ABB RAPID module: test02_001.prg

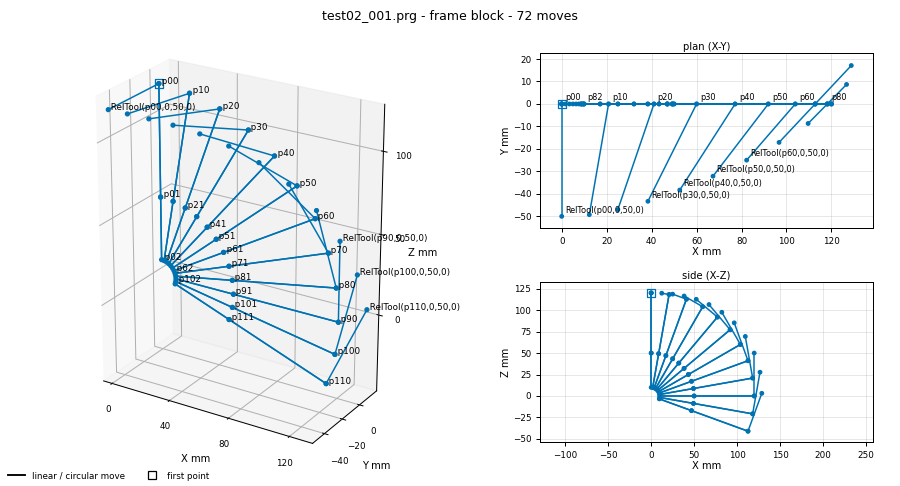
[picture p0: tool path of test02_001.prg in frame block, 72 of 87 moves have a stored position in this frame; points joined in program order, loops and branches not executed]
MODULE MainModule

	! test02_001

	! variables
	TASK PERS tooldata drill := [FALSE, [[300,-260,280], [0,0,0,1]], [1,[0,0,0.001],[1,0,0,0],0,0,0]];
	TASK PERS wobjdata block := [TRUE, TRUE, "", [[0,0,150], [1,0,0,0]], [[0,0,0], [1,0,0,0]]];
	TASK PERS speeddata rate := [3, 500, 5000, 1000];

	! targets
	VAR jointtarget j0 := [[-90,0,0,90,90,0], [9E9,9E9,9E9,9E9,9E9,9E9]];
	VAR jointtarget j1 := [[-41,0,0,0,90,0], [9E9,9E9,9E9,9E9,9E9,9E9]];
	VAR robtarget p00 := [[2.20429143688028E-14,0,120], [0,1,0,-9.18454765366783E-17], [0,0,0,0], [9E9,9E9,9E9,9E9,9E9,9E9]];
	VAR robtarget p01 := [[9.18454765366783E-15,0,50], [0,1,0,-9.18454765366783E-17], [0,0,0,0], [9E9,9E9,9E9,9E9,9E9,9E9]];
	VAR robtarget p02 := [[1.83690953073357E-15,0,10], [0,1,0,-9.18454765366783E-17], [0,0,0,0], [9E9,9E9,9E9,9E9,9E9,9E9]];
	VAR robtarget p10 := [[20.8377813200316,-1.2490009027033E-15,118.176930361465], [0.00759612349389579,0.992403876506124,-0.0868240888334661,-0.086824088833467], [0,0,0,0], [9E9,9E9,9E9,9E9,9E9,9E9]];
	VAR robtarget p11 := [[8.68240888334652,-5.20417042793042E-16,49.2403876506104], [0.00759612349389579,0.992403876506124,-0.0868240888334661,-0.086824088833467], [0,0,0,0], [9E9,9E9,9E9,9E9,9E9,9E9]];
	VAR robtarget p12 := [[1.7364817766693,-1.04083408558608E-16,9.84807753012208], [0.00759612349389579,0.992403876506124,-0.0868240888334661,-0.086824088833467], [0,0,0,0], [9E9,9E9,9E9,9E9,9E9,9E9]];
	VAR robtarget p20 := [[41.0424171990802,-1.66533453693773E-15,112.763114494309], [0.0301536896070456,0.969846310392959,-0.171010071662836,-0.171010071662835], [0,0,0,0], [9E9,9E9,9E9,9E9,9E9,9E9]];
	VAR robtarget p21 := [[17.1010071662834,-6.93889390390723E-16,46.9846310392954], [0.0301536896070456,0.969846310392959,-0.171010071662836,-0.171010071662835], [0,0,0,0], [9E9,9E9,9E9,9E9,9E9,9E9]];
	VAR robtarget p22 := [[3.42020143325669,-1.38777878078145E-16,9.39692620785909], [0.0301536896070456,0.969846310392959,-0.171010071662836,-0.171010071662835], [0,0,0,0], [9E9,9E9,9E9,9E9,9E9,9E9]];
	VAR robtarget p30 := [[60.0000000000001,-6.66133814775094E-15,103.923048454133], [0.0669872981077809,0.933012701892218,-0.249999999999999,-0.25], [0,0,0,0], [9E9,9E9,9E9,9E9,9E9,9E9]];
	VAR robtarget p31 := [[25,-2.77555756156289E-15,43.3012701892219], [0.0669872981077809,0.933012701892218,-0.249999999999999,-0.25], [0,0,0,0], [9E9,9E9,9E9,9E9,9E9,9E9]];
	VAR robtarget p32 := [[5,-5.55111512312578E-16,8.66025403784439], [0.0669872981077809,0.933012701892218,-0.249999999999999,-0.25], [0,0,0,0], [9E9,9E9,9E9,9E9,9E9,9E9]];
	VAR robtarget p40 := [[77.1345131623847,6.66133814775094E-15,91.9253331742773], [0.116977778440511,0.883022221559491,-0.32139380484327,-0.32139380484327], [0,0,0,0], [9E9,9E9,9E9,9E9,9E9,9E9]];
	VAR robtarget p41 := [[32.139380484327,2.77555756156289E-15,38.3022221559489], [0.116977778440511,0.883022221559491,-0.32139380484327,-0.32139380484327], [0,0,0,0], [9E9,9E9,9E9,9E9,9E9,9E9]];
	VAR robtarget p42 := [[6.4278760968654,5.55111512312578E-16,7.66044443118978], [0.116977778440511,0.883022221559491,-0.32139380484327,-0.32139380484327], [0,0,0,0], [9E9,9E9,9E9,9E9,9E9,9E9]];
	VAR robtarget p50 := [[91.9253331742774,9.99200722162641E-15,77.1345131623847], [0.17860619515673,0.82139380484327,-0.383022221559489,-0.383022221559489], [0,0,0,0], [9E9,9E9,9E9,9E9,9E9,9E9]];
	VAR robtarget p51 := [[38.3022221559489,4.16333634234434E-15,32.139380484327], [0.17860619515673,0.82139380484327,-0.383022221559489,-0.383022221559489], [0,0,0,0], [9E9,9E9,9E9,9E9,9E9,9E9]];
	VAR robtarget p52 := [[7.66044443118978,8.32667268468867E-16,6.4278760968654], [0.17860619515673,0.82139380484327,-0.383022221559489,-0.383022221559489], [0,0,0,0], [9E9,9E9,9E9,9E9,9E9,9E9]];
	VAR robtarget p60 := [[103.923048454133,1.33226762955019E-14,60], [0.25,0.75,-0.433012701892219,-0.433012701892219], [0,0,0,0], [9E9,9E9,9E9,9E9,9E9,9E9]];
	VAR robtarget p61 := [[43.3012701892219,5.55111512312578E-15,25], [0.25,0.75,-0.433012701892219,-0.433012701892219], [0,0,0,0], [9E9,9E9,9E9,9E9,9E9,9E9]];
	VAR robtarget p62 := [[8.66025403784439,1.11022302462516E-15,5], [0.25,0.75,-0.433012701892219,-0.433012701892219], [0,0,0,0], [9E9,9E9,9E9,9E9,9E9,9E9]];
	VAR robtarget p70 := [[112.763114494309,6.66133814775094E-15,41.0424171990802], [0.328989928337166,0.671010071662834,-0.469846310392954,-0.469846310392954], [0,0,0,0], [9E9,9E9,9E9,9E9,9E9,9E9]];
	VAR robtarget p71 := [[46.9846310392954,2.77555756156289E-15,17.1010071662834], [0.328989928337166,0.671010071662834,-0.469846310392954,-0.469846310392954], [0,0,0,0], [9E9,9E9,9E9,9E9,9E9,9E9]];
	VAR robtarget p72 := [[9.39692620785909,5.55111512312578E-16,3.42020143325669], [0.328989928337166,0.671010071662834,-0.469846310392954,-0.469846310392954], [0,0,0,0], [9E9,9E9,9E9,9E9,9E9,9E9]];
	VAR robtarget p80 := [[118.176930361465,3.7470027081099E-15,20.8377813200317], [0.413175911166535,0.586824088833465,-0.492403876506104,-0.492403876506104], [0,0,0,0], [9E9,9E9,9E9,9E9,9E9,9E9]];
	VAR robtarget p81 := [[49.2403876506104,1.56125112837913E-15,8.68240888334652], [0.413175911166535,0.586824088833465,-0.492403876506104,-0.492403876506104], [0,0,0,0], [9E9,9E9,9E9,9E9,9E9,9E9]];
	VAR robtarget p82 := [[9.84807753012208,3.12250225675825E-16,1.7364817766693], [0.413175911166535,0.586824088833465,-0.492403876506104,-0.492403876506104], [0,0,0,0], [9E9,9E9,9E9,9E9,9E9,9E9]];
	VAR robtarget p90 := [[120,-8.99826150854451E-31,-1.46952762458685E-14], [0.5,0.5,-0.5,-0.5], [0,0,0,0], [9E9,9E9,9E9,9E9,9E9,9E9]];
	VAR robtarget p91 := [[50,-3.74927562856021E-31,-6.12303176911188E-15], [0.5,0.5,-0.5,-0.5], [0,0,0,0], [9E9,9E9,9E9,9E9,9E9,9E9]];
	VAR robtarget p92 := [[10,-7.49855125712043E-32,-1.22460635382238E-15], [0.5,0.5,-0.5,-0.5], [0,0,0,0], [9E9,9E9,9E9,9E9,9E9,9E9]];
	VAR robtarget p100 := [[118.176930361465,-1.66533453693773E-15,-20.8377813200316], [0.586824088833465,0.413175911166535,-0.492403876506104,-0.492403876506104], [0,0,0,0], [9E9,9E9,9E9,9E9,9E9,9E9]];
	VAR robtarget p101 := [[49.2403876506104,-6.93889390390723E-16,-8.68240888334652], [0.586824088833465,0.413175911166535,-0.492403876506104,-0.492403876506104], [0,0,0,0], [9E9,9E9,9E9,9E9,9E9,9E9]];
	VAR robtarget p102 := [[9.84807753012208,-1.38777878078145E-16,-1.7364817766693], [0.586824088833465,0.413175911166535,-0.492403876506104,-0.492403876506104], [0,0,0,0], [9E9,9E9,9E9,9E9,9E9,9E9]];
	VAR robtarget p110 := [[112.763114494309,-3.33066907387547E-15,-41.0424171990803], [0.671010071662834,0.328989928337166,-0.469846310392954,-0.469846310392954], [0,0,0,0], [9E9,9E9,9E9,9E9,9E9,9E9]];
	VAR robtarget p111 := [[46.9846310392954,-1.38777878078145E-15,-17.1010071662834], [0.671010071662834,0.328989928337166,-0.469846310392954,-0.469846310392954], [0,0,0,0], [9E9,9E9,9E9,9E9,9E9,9E9]];
	VAR robtarget p112 := [[9.39692620785908,-2.77555756156289E-16,-3.42020143325669], [0.671010071662834,0.328989928337166,-0.469846310392954,-0.469846310392954], [0,0,0,0], [9E9,9E9,9E9,9E9,9E9,9E9]];

	! drilling instructions
	PROC main()
		ConfL\Off;
		SingArea\Wrist;

		TPWrite("This is: test02_001");
		TPWrite("Check block and drill");
		MoveAbsJ j0, v100, z5, tool0;
		MoveAbsJ j1, v100, z5, tool0;

		TPWrite("Drilling hole 1 of 12!");
		MoveL p00, v100, z30, drill\WObj:=block;
		MoveL p01, v100, z5, drill\WObj:=block;
		MoveL p02, rate, fine, drill\WObj:=block;
		MoveL p01, rate, fine, drill\WObj:=block;
		MoveL p00, v100, z30, drill\WObj:=block;
		MoveL RelTool(p00, 0, 50, 0), v100, z5, drill\WObj:=block;
		MoveAbsJ CalcJointT(RelTool(p10, 0, 50, 0), drill\WObj:=block), v100, z5, drill\WObj:=block;

		TPWrite("Drilling hole 2 of 12!");
		MoveL p10, v100, z30, drill\WObj:=block;
		MoveL p11, v100, z5, drill\WObj:=block;
		MoveL p12, rate, fine, drill\WObj:=block;
		MoveL p11, rate, fine, drill\WObj:=block;
		MoveL p10, v100, z30, drill\WObj:=block;
		MoveL RelTool(p10, 0, 50, 0), v100, z5, drill\WObj:=block;
		MoveAbsJ CalcJointT(RelTool(p20, 0, 50, 0), drill\WObj:=block), v100, z5, drill\WObj:=block;

		TPWrite("Drilling hole 3 of 12!");
		MoveL p20, v100, z30, drill\WObj:=block;
		MoveL p21, v100, z5, drill\WObj:=block;
		MoveL p22, rate, fine, drill\WObj:=block;
		MoveL p21, rate, fine, drill\WObj:=block;
		MoveL p20, v100, z30, drill\WObj:=block;
		MoveL RelTool(p20, 0, 50, 0), v100, z5, drill\WObj:=block;
		MoveAbsJ CalcJointT(RelTool(p30, 0, 50, 0), drill\WObj:=block), v100, z5, drill\WObj:=block;

		TPWrite("Drilling hole 4 of 12!");
		MoveL p30, v100, z30, drill\WObj:=block;
		MoveL p31, v100, z5, drill\WObj:=block;
		MoveL p32, rate, fine, drill\WObj:=block;
		MoveL p31, rate, fine, drill\WObj:=block;
		MoveL p30, v100, z30, drill\WObj:=block;
		MoveL RelTool(p30, 0, 50, 0), v100, z5, drill\WObj:=block;
		MoveAbsJ CalcJointT(RelTool(p40, 0, 50, 0), drill\WObj:=block), v100, z5, drill\WObj:=block;

		TPWrite("Drilling hole 5 of 12!");
		MoveL p40, v100, z30, drill\WObj:=block;
		MoveL p41, v100, z5, drill\WObj:=block;
		MoveL p42, rate, fine, drill\WObj:=block;
		MoveL p41, rate, fine, drill\WObj:=block;
		MoveL p40, v100, z30, drill\WObj:=block;
		MoveL RelTool(p40, 0, 50, 0), v100, z5, drill\WObj:=block;
		MoveAbsJ CalcJointT(RelTool(p50, 0, 50, 0), drill\WObj:=block), v100, z5, drill\WObj:=block;

		TPWrite("Drilling hole 6 of 12!");
		MoveL p50, v100, z30, drill\WObj:=block;
		MoveL p51, v100, z5, drill\WObj:=block;
		MoveL p52, rate, fine, drill\WObj:=block;
		MoveL p51, rate, fine, drill\WObj:=block;
		MoveL p50, v100, z30, drill\WObj:=block;
		MoveL RelTool(p50, 0, 50, 0), v100, z5, drill\WObj:=block;
		MoveAbsJ CalcJointT(RelTool(p60, 0, 50, 0), drill\WObj:=block), v100, z5, drill\WObj:=block;

		TPWrite("Drilling hole 7 of 12!");
		MoveL p60, v100, z30, drill\WObj:=block;
		MoveL p61, v100, z5, drill\WObj:=block;
		MoveL p62, rate, fine, drill\WObj:=block;
		MoveL p61, rate, fine, drill\WObj:=block;
		MoveL p60, v100, z30, drill\WObj:=block;
		MoveL RelTool(p60, 0, 50, 0), v100, z5, drill\WObj:=block;
		MoveAbsJ CalcJointT(RelTool(p70, 0, 50, 0), drill\WObj:=block), v100, z5, drill\WObj:=block;

		TPWrite("Drilling hole 8 of 12!");
		MoveL p70, v100, z30, drill\WObj:=block;
		MoveL p71, v100, z5, drill\WObj:=block;
		MoveL p72, rate, fine, drill\WObj:=block;
		MoveL p71, rate, fine, drill\WObj:=block;
		MoveL p70, v100, z30, drill\WObj:=block;
		MoveL RelTool(p70, 0, 50, 0), v100, z5, drill\WObj:=block;
		MoveAbsJ CalcJointT(RelTool(p80, 0, 50, 0), drill\WObj:=block), v100, z5, drill\WObj:=block;

		TPWrite("Drilling hole 9 of 12!");
		MoveL p80, v100, z30, drill\WObj:=block;
		MoveL p81, v100, z5, drill\WObj:=block;
		MoveL p82, rate, fine, drill\WObj:=block;
		MoveL p81, rate, fine, drill\WObj:=block;
		MoveL p80, v100, z30, drill\WObj:=block;
		MoveL RelTool(p80, 0, 50, 0), v100, z5, drill\WObj:=block;
		MoveAbsJ CalcJointT(RelTool(p90, 0, 50, 0), drill\WObj:=block), v100, z5, drill\WObj:=block;

		TPWrite("Drilling hole 10 of 12!");
		MoveL p90, v100, z30, drill\WObj:=block;
		MoveL p91, v100, z5, drill\WObj:=block;
		MoveL p92, rate, fine, drill\WObj:=block;
		MoveL p91, rate, fine, drill\WObj:=block;
		MoveL p90, v100, z30, drill\WObj:=block;
		MoveL RelTool(p90, 0, 50, 0), v100, z5, drill\WObj:=block;
		MoveAbsJ CalcJointT(RelTool(p100, 0, 50, 0), drill\WObj:=block), v100, z5, drill\WObj:=block;

		TPWrite("Drilling hole 11 of 12!");
		MoveL p100, v100, z30, drill\WObj:=block;
		MoveL p101, v100, z5, drill\WObj:=block;
		MoveL p102, rate, fine, drill\WObj:=block;
		MoveL p101, rate, fine, drill\WObj:=block;
		MoveL p100, v100, z30, drill\WObj:=block;
		MoveL RelTool(p100, 0, 50, 0), v100, z5, drill\WObj:=block;
		MoveAbsJ CalcJointT(RelTool(p110, 0, 50, 0), drill\WObj:=block), v100, z5, drill\WObj:=block;

		TPWrite("Drilling hole 12 of 12!");
		MoveL p110, v100, z30, drill\WObj:=block;
		MoveL p111, v100, z5, drill\WObj:=block;
		MoveL p112, rate, fine, drill\WObj:=block;
		MoveL p111, rate, fine, drill\WObj:=block;
		MoveL p110, v100, z30, drill\WObj:=block;
		MoveL RelTool(p110, 0, 50, 0), v100, z5, drill\WObj:=block;

		TPWrite("Resetting axes...");
		MoveAbsJ j1, v100, z5, tool0;
		MoveAbsJ j0, v100, z5, tool0;

		Stop;
	ENDPROC

ENDMODULE
